// TIA Portal V20 export
// export: Created 2025-12-01T14:57:44.562273Z, ExportSetting None, DisplayName Totally Integrated Automation Portal, DisplayVersion V20 Update 3, DisplayName TIA Portal Openness, DisplayVersion V20 Update 3, DisplayName TIA Portal Version Control Interface, DisplayVersion V20 Update 3, DisplayName STEP 7 Professional, DisplayVersion V20 Update 3, DisplayName STEP 7 Safety, DisplayVersion V20 Update 2, DisplayName WinCC Basic/Comfort/Advanced, DisplayVersion V20 Update 3, DisplayName WinCC Professional, DisplayVersion V20 Update 3, DisplayName WinCC Unified, DisplayVersion V20 Update 3
FUNCTION "FC570_Leer_Zona_Entradas" : Void   // FC570, STL
{ S7_Optimized_Access := 'FALSE' }
// stored: AutoNumber false
   VAR_INPUT
      Inicio_Zona : UInt;   // Numero de scanner sobre el que se realiza la busqueda
      Long_Zona : UInt;
   END_VAR
   VAR_OUTPUT
      Datos_Zona : Any;
   END_VAR
   VAR_TEMP
      Guardar_AR2 : DWord;
      P_Inicio_Datos : DWord;
      P_Any_Datos : Any;
      LongRegistro : UInt;
      ValorReturn : Int;
      Relleno : Byte;
   END_VAR
BEGIN

NETWORK
TITLE = Inicializar Variables
//////////////////////////////////////////////////////////////////////////
/// - Datos del DB a leer

      L     #Long_Zona;
      T     #LongRegistro;


//////////////////////////////////////////////////////////////////////////
/// - Inicilizar Registro de Salida

      L     0;
      T     #Relleno;

      CALL  FILL
      ( BVAL    := #Relleno,
        RET_VAL := #ValorReturn,
        BLK     := #Datos_Zona
      );



NETWORK
TITLE = Posicionarse en el Registro
//////////////////////////////////////////////////////////////////////////
/// - Calculo de la posicion del registro

// primero nos posicionamos en el primer elemento de la fifo

      L     #Inicio_Zona;
      SLD   3;
      T     #P_Inicio_Datos;




NETWORK
TITLE = Transferenica del Registro
//////////////////////////////////////////////////////////////////////////
/// - Calculo del Puntero Any de los Datos
sacar_datos:NOP   0;
      TAR2  #Guardar_AR2;  // - Guardar el Puntero AR2

      LAR2  P##P_Any_Datos;  // - Direccion del Puntero Any
      L     B#16#10;  //   10H para S7
      T     LB [AR2, P#0.0];
      L     B#16#2;  //   Tipo de Datos (BYTE)
      T     LB [AR2, P#1.0];
      L     #LongRegistro;  //   Longitud de la Estructura
      T     LW [AR2, P#2.0];
      L     0;  //   Numero de DB
      T     LW [AR2, P#4.0];
      L     #P_Inicio_Datos;  //   Direccion de Inicio
      T     LD [AR2, P#6.0];
      L     B#16#81;  //   El Area de Memoria = DB
      T     LB [AR2, P#6.0];

      LAR2  #Guardar_AR2;  // - Recuperar el Puntero AR2

//////////////////////////////////////////////////////////////////////////
/// - Transferencia de los Datos a Leer

      CALL  BLKMOV
      ( SRCBLK  := #P_Any_Datos,
        RET_VAL := #ValorReturn,
        DSTBLK  := #Datos_Zona
      );

      L     #ValorReturn;  // - Comprobar que se ha leido el registro
      L     0;
      <>I;
      JC    Error_LecturaDelRegisto;


//////////////////////////////////////////////////////////////////////////
/// - Fin de la Lectura del Registro

      BE;  // - Finalizar bloque



NETWORK
TITLE = Errores en el Sistema de Lectura
//////////////////////////////////////////////////////////////////////////
/// - Numero De Maximo de Registros Sobrepasado

Error_MaxRegistros:NOP   0;
      BE;  // - Finalizar bloque

////////////////////////////////////////////////////
/// - Error a Leer el Registro

Error_LecturaDelRegisto:NOP   0;
      BE;  // - Finalizar bloque


END_FUNCTION
